TYPE U_TRIGGER_STATE :
UNION
  stState              : ARRAY[1..MAX_TRIGGER_BOX] OF ST_STATE_TRIGGER;

  byState    AT %i*   : ARRAY[1..MAX_TRIGGER_BOX] OF
                        ARRAY[1..SIZEOF(ST_STATE_TRIGGER)] OF BYTE;
END_UNION
END_TYPE

(* stored: Version 1.1.0.1
   DUT U_TRIGGER_STATE: Id {b8dbc0bf-bd9b-4e0a-8637-87a8e34441c6} *)
